// TIA Portal V17 export
// export: Created 2025-03-07T09:17:49.9515606Z, ExportSetting WithDefaults, DisplayName Totally Integrated Automation Portal, DisplayVersion V17 Update 8, DisplayName TIA Portal Openness, DisplayVersion V17 Update 8, DisplayName TIA Portal Version Control Interface, DisplayVersion V17, DisplayName SINAMICS Startdrive Advanced, DisplayVersion V17 SP2, DisplayName SINAMICS Startdrive G110M, G120, G120C, G120D, G120P, G115D, DisplayVersion V17 SP2, DisplayName SINAMICS Startdrive G130, G150, S120, S150, SINAMICS MV, S210, DisplayVersion V17 SP2, DisplayName STEP 7 Professional, DisplayVersion V17 Update 8, DisplayName SINUMERIK ONE STEP 7 Toolbox, DisplayVersion V17 Update 12, DisplayName SINUMERIK 840D sl STEP 7 Toolbox, DisplayVersion V17 Update 12, DisplayName STEP 7 Safety, DisplayVersion V17 Update 6, DisplayName WinCC Advanced, DisplayVersion V17 Update 8
DATA_BLOCK "DB2120_MPP_ITC_IPC"   // DB2120
{ S7_Optimized_Access := 'FALSE'; DB_Accessible_From_OPC_UA := 'FALSE' }
AUTHOR : ETXETAR
VERSION : 1.0
// stored: AutoNumber false, DBAccessibleFromOPCUA false, DBAccessibleFromWebserver true, IsOnlyStoredInLoadMemory false, IsWriteProtectedInAS false
   VAR RETAIN
      INPUT_CONTROL_ON : Bool;   // INPUT CONTROL ON
      INPUT_MACHINE_OFF : Bool;   // INPUT MACHINE OFF
      CONTROL_ON : Bool;   // CONTROL ON
      CONTROL_ON_DELAYED : Bool;   // CONTROL ON DELAYED
      CONTROL_ON_PULSE : Bool;   // CONTROL ON PULSE
      CONTROL_OFF3_DELAYED : Bool;   // MACHINE OFF DELAYED / CONTROL OFF3 DELAYED
      CONTROL_ON_OFF_DELAYED : Bool;   // MACHINE OFF DELAYED / CONTROL ON/OFF DELAYED
      MACHINE_ON : Bool;   // MACHINE ON
      MACHINE_ON_DELAYED : Bool;   // MACHINE ON DELAYED
      MACHINE_OFF_DELAYED : Bool;   // MACHINE OFF DELAYED
      MACHINE_ON_DELAYED_PULSE : Bool;   // MACHINE ON DELAYED PULSE
      MACHINE_ON_DELAYED_AUX : Bool;   // MACHINE ON DELAYED AUXILIARY
      MACH_ON_DEL_PNEU_ON : Bool;   // CRM + HYD + PNEUMATIC ON / MACHINE ON DELAYED PNEUMATIC IN SERVICE
      MACH_STOP_SERV_ENABLED : Bool;   // MACHINE STOP SERVICES DELAYED ENABLED
      MACH_STOP_SERV_DELAY_1 : Bool;   // MACHINE STOP SERVICES DELAYED 1
      MACH_STOP_SERV_DELAY_2 : Bool;   // MACHINE STOP SERVICES DELAYED 2
      MPP_MAIN_PANEL_ACTIVE : Bool;   // MPP MAIN PANEL ACTIVE
      ITC_1_ACTIVE : Bool;   // TCU 1 ACTIVE / ITC 1 ACTIVE
      HT10_ACTIVE : Bool;   // HT8 ACTIVE / HT10 ACTIVE
      AXES_OVERRIDE : Byte;   // AXES OVERRIDE
      AXES_OVERRIDE_DECIMAL : Byte;   // RESERVED / AXES OVERRIDE VALUE IN DECIMAL
      SPINDLES_OVERRIDE : Byte;   // SPINDLES OVERRIDE
      OVERRIDE_ZERO : Bool;   // OVERRIDE ZERO
      OVERRIDE_LOWER_THAN_80 : Bool;   // OVERRIDE LOWER THAN 80
      OVERRIDE_100 : Bool;   // OVERRIDE 100
      START_SERVICES_GLOBAL : Bool;   // START SERVICES GLOBAL
      START_CYCLE_GLOBAL : Bool;   // START CYCLE GLOBAL
      RETURN_HOME_POSITION_BY_OPERATOR : Bool;   // RETURN HOME POSITION BY OPERATOR
      RETURN_HOME_POSITION_BY_OPERATOR_AUX_1 : Bool;   // RETURN HOME POSITION BY OPERATOR / RETURN HOME POSITION BY OPERATOR AUXILIARY 1
      RETURN_HOME_POSITION_BY_OPERATOR_AUX_2 : Bool;   // RETURN HOME POSITION BY OPERATOR / RETURN HOME POSITION BY OPERATOR AUXILIARY 2
      RETURN_HOME_POSITION_FROM_MPP_PANEL : Bool;   // RETURN HOME POSITION FROM MPP PANNEL / RETURN HOME POSITION FROM MPP PANEL
      RETURN_HOME_POSITION_FROM_AUX_PANEL : Bool;   // RETURN HOME POSITION FROM AUX PANEL
      RETURN_HOME_POSITION_PULSE : Bool;   // END OF CYCLE TOGGLE AUXILIAR FUNCTION / RETURN HOME POSITION PULSE
      RESET_FAULTS : Bool;   // RESET FAULT / RESET FAULTS
      RESET_FAULTS_PULSE : Bool;   // RESET FAULT PULSE / RESET FAULTS PULSE
      RESET_FAULTS_GLOBAL : Bool;   // RESET FAULTS GLOBAL
      RESET_FAULTS_AUX : Bool;   // AUXILIARY RESET FAULT / RESET FAULTS AUXILIARY
      STOP_SERVICES_GLOBAL : Bool;   // STOP SERVICES GLOBAL
      STOP_END_OF_CYCLE_REQUEST : Bool;   // STOP END OF CYCLE REQUEST
      AUX_STOP_END_CYCLE_REQUEST : Bool;   // AUX STOP END CYCLE REQUEST
      STOP_END_OF_CYCLE_FROM_MPP_PANEL : Bool;   // END OF CYCLE FROM MPP PANNEL / STOP END OF CYCLE FROM MPP PANEL
      STOP_END_OF_CYCLE_FROM_AUX_PANEL : Bool;   // END OF CYCLE FROM AUX PANNEL / STOP END OF CYCLE FROM AUX PANEL
      STOP_END_OF_CYCLE_BY_OPERATOR : Bool;   // STOP END OF CYCLE BY OPERATOR
      STOP_END_OF_CYCLE_BY_OPERATOR_AUX_1 : Bool;   // STOP END OF CYCLE BY OPERATOR / STOP END OF CYCLE BY OPERATOR AUXILIARY 1
      STOP_END_OF_CYCLE_BY_OPERATOR_AUX_2 : Bool;   // STOP END OF CYCLE BY OPERATOR / STOP END OF CYCLE BY OPERATOR AUXILIARY 2
      STOP_END_OF_CYCLE_PULSE : Bool;   // END OF CYCLE BY OPERATOR ACTIVE / STOP END OF CYCLE PULSE
      IMMEDIATE_STOP_BY_OPERATOR : Bool;   // IMMEDIATY STOP BY OPERATOR / IMMEDIATE STOP BY OPERATOR
      IMMEDIATE_STOP_BY_OPERATOR_AUX : Bool;   // IMMEDIATY STOP BY OPERATOR / IMMEDIATE STOP BY OPERATOR AUXILIARY
      IMMEDIATE_STOP_GLOBAL : Bool;   // IMMEDIATE STOP GLOBAL
      SAFETY_DOORS_NOT_CLOSED : Bool;   // PILZS GATES NOT CLOSED / SAFETY DOORS NOT CLOSED
      ANY_SAFETY_DOOR_UNLOCK_COMAND : Bool;   // ANY SAFETY DOOR UNLOCK COMMAND
      ANY_SAFETY_DOOR_UNLOCK : Bool;   // ANY SAFETY DOOR UNLOCK
      BIMANUAL_F1_UNLOAD_PARTS_CONDITIONS : Bool;   // BIMANUAL FIXTURE 1 UNLOAD PARTS CONDITIONS
      BIMANUAL_F2_UNLOAD_PARTS_CONDITIONS : Bool;   // BIMANUAL FIXTURE 2 UNLOAD PARTS CONDITIONS
      TIMER_CONTROL_ON : TON_TIME;   // CONTROL ON TIMER
      TIMER_MACHINE_ON : TON_TIME;   // MACHINE ON TIMER
      TIMER_MACHINE_OFF : TOF_TIME;   // MACHINE OFF TIMER
      TIMER_MACH_STOP_SERV_DELAY : TON_TIME;   // MACHINE STOP SERVICES TIMER
      TIMER_BIMANUAL_CYCLE_START : TON_TIME;   // BIMANUAL CYCLE START TIMER
      TIMER_CONTROL_OFF : TOF_TIME;   // CONTROL OFF TIMER
      TIMER_CONTROL_OFF3 : TOF_TIME;   // CONTROL OFF3 TIMER
      TIMER_CONTROL_ON_OFF : TOF_TIME;   // CONTROL ON/OFF TIMER
   END_VAR
BEGIN
   TIMER_CONTROL_ON.PT := T#3s;
   TIMER_MACHINE_ON.PT := T#2s;
   TIMER_MACHINE_OFF.PT := T#3s;
   TIMER_BIMANUAL_CYCLE_START.PT := T#2s;
   TIMER_CONTROL_OFF.PT := T#1s;
   TIMER_CONTROL_OFF3.PT := T#5s;
   TIMER_CONTROL_ON_OFF.PT := T#6s;
END_DATA_BLOCK
